TYPE ST_AutoAddsBoxesCommand EXTENDS ST_CommandBasic :
STRUCT
END_STRUCT
END_TYPE

(* stored: Version 1.1.0.1, ProductVersion 3.1.4024.13
   DUT ST_AutoAddsBoxesCommand: Id {f93407c2-0636-4329-b8b9-0847a70a42de} *)
